(* -----------------------------------------------------------------------------
| This sample has been supplied by Beckhoff As-Is and is intended only as an   |
| example implementation. Functionality is not guaranteed.                     |
----------------------------------------------------------------------------- *)

PROGRAM MAIN
VAR
	fbStateMachine : FB_StateMachine;
	fbVisuSim : FB_VisuSim;
END_VAR

(* -----------------------------------------------------------------------------
| This sample has been supplied by Beckhoff As-Is and is intended only as an   |
| example implementation. Functionality is not guaranteed.                     |
----------------------------------------------------------------------------- *)

fbStateMachine(
	bStart:= GVL.bStart, 
	bStop:= GVL.bStop, 
	bBottle:= GVL.bBottle,	 
);

GVL.bConveyor := fbStateMachine.bConveyor;
GVL.bWater := fbStateMachine.bWater;
GVL.bMint := fbStateMachine.bMint;	
GVL.bCorking := fbStateMachine.bCorking;

(* Visu and Simulation *)
fbVisuSim(bConveyor:= GVL.bConveyor);
GVL.bBottle := fbVisuSim.bBottle;

END_PROGRAM

(* stored: Version 1.1.0.1, ProductVersion 3.1.4024.12
   POU MAIN: Id {97e09f56-a846-45b7-b746-7c26db2ee647}, SpecialFunc None *)
